Staubli VAL3: onExit.pgx

program onExit()
begin
  //
  //  Kill it
  //
  // relaod the template session
  call saveData:changeSession("template")
  // exit
  logMsg("[KERNEL] INTERFACE:Quit")
  cycleStatus:nInterfaceToSV=1
  //
  //
end
